Yaskawa INFORM job: DATAHIGHWAY.JBI

/JOB
//NAME DATAHIGHWAY
//POS
///NPOS 0,0,0,0,0,0
//INST
///DATE 2026/05/04 14:59
///ATTR SC,RW
///GROUP1 RB1
NOP
SKILLSND SL5 "barcodeScan"
SKILLSND SL5 "fetchRecipe"
END
